FUNCTION_BLOCK UNSCALE (* Integer Unscaling of an integer input of 0-100% *)
  (* Standard: 61499-1 *)
  (* Version 0.0, 2004-09-01, JHC, Rockwell Automation *)
  (* Compiler header: package fb.rt.process; *)
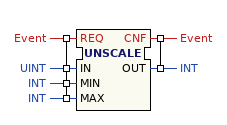
  EVENT_INPUT
    REQ WITH IN, MIN, MAX; (* Normal Execution Request *)
  END_EVENT
  EVENT_OUTPUT
    CNF WITH OUT; (* Execution Confirmation *)
  END_EVENT
  VAR_INPUT
    IN : UINT; (* Scaled Input, 0-100% *)
    MIN : INT; (* OUT value corresponding to IN=0 *)
    MAX : INT; (* OUT value corrsponding to IN=100% *)
  END_VAR
  VAR_OUTPUT
    OUT : INT; (* Unscaled Output corresponding to IN value *)
  END_VAR
  ALGORITHM REQ IN ST: (* Unscaling algorithm *)
OUT := MIN + (MAX-MIN)*IN/100;
CNF.serviceEvent(this);
  END_ALGORITHM
END_FUNCTION_BLOCK
